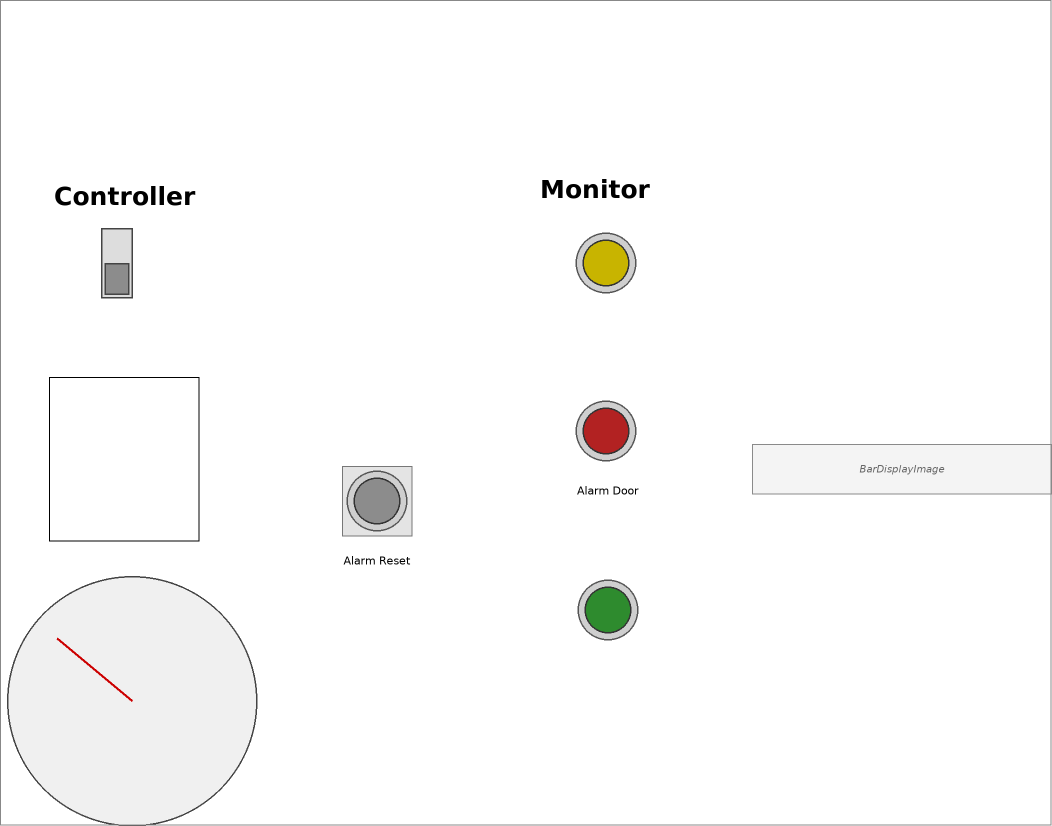
VISUALIZATION VisuMain  // 1052x826
    Lamp1 (571,228 70x70), variable: GVL_Var.bLight, style: Lamp-Lamp1-Yellow
    DipSwitch (82,228 70x70), variable: GVL_Var.bDoorOpen, behaviour: TOGGLE, style: Switch-DipSwitch-Gray
    Rectangle (49,377 150x164)
        toggle GVL_Var.bDoorOpen
    Lamp1 (571,396 70x70), variable: GVL_Var.bAlarmOut, style: Lamp-Lamp1-Red
    Label (533,476 150x30), "Alarm Door"
    Label (27,163 204x66), "Controller"
    Label (520,174 150x30), "Monitor"
    PushSwitch (342,466 70x70), variable: GVL_Var.bAlarmReset, behaviour: TOGGLE, style: Switch-PushSwitch-Gray
    Label (302,546 150x30), "Alarm Reset"
    Meter360 (7,576 250x250), value: GVL_Var.fTempSet, style: Meter-Meter360-Gray, scale format: %.0f, scale 0..20
    Lamp1 (573,575 70x70), variable: GVL_Var.bCompressor, style: Lamp-Lamp1-Green
    BarDisplayImage (752,444 300x50), value: GVL_Var.fTempActual, style: BarDisplayImage-Gray, scale format: %.1f, scale 0..24
END_VISUALIZATION

(* stored: Version 1.1.0.1, ProductVersion 3.1.4026.18
   Visu VisuMain: Id {c8f5eb35-6d66-4bb4-b9c9-5612d360c93a} *)
